# EPICS substitutions: db/Beckhoff_7XXX/ecmcEL7037_CSP.substitutions
file "ecmcEL7037_CSP-chX.template"
{
  pattern {CH_ID}
          {01   }
}

file "ecmcEL5101-chX.template"
{
  pattern {CH_ID}
          {01   }
}
